{attribute addProperty BoxType "EK1100-0000-0018"}
{attribute addProperty Id "Beckhoff_EL29xxEK1122Beckhoff_EL29xxEK1122_E909BF84162A_0001_EL2911_0000_0016EL2911_049EC81322027.5A_0002_EL2912_0000_0016EL2912_398D870922828.5"}
{attribute addProperty CRC "1275110990"}
{attribute addProperty SizeInBites "464"}
{attribute addProperty SizeInBytes "58"}
TYPE Beckhoff_EL29xx_4C00A64E EXTENDS EK1100_179A0949 :
STRUCT
	{attribute addProperty Name "Beckhoff_EL29xxEK1122"}
	Beckhoff_EL29xxEK1122 : Beckhoff_EL29xxEK1122_E909BF84;
	{attribute addProperty Name "A_0001_EL2911_0000_0016"}
	A_0001_EL2911_0000_0016 : EL2911_049EC813;
	{attribute addProperty Name "A_0002_EL2912_0000_0016"}
	A_0002_EL2912_0000_0016 : EL2912_398D8709;
END_STRUCT
END_TYPE

(* stored: Version 1.2.0.0, ProductVersion 3.1.4024.9
   DUT Beckhoff_EL29xx_4C00A64E: Id {58c8d1bd-59a2-4b41-acb7-ebd02094810a} *)
